{attribute 'pack_mode' := '2'}
TYPE U_XTS_TRANSPORT_CTRL :
UNION
  stCtrl              : ST_XTS_TRANSPORT_CTRL;
  byCtrl    AT %I*    : ARRAY[1..SIZEOF(ST_XTS_TRANSPORT_CTRL)] OF BYTE;
END_UNION
END_TYPE

(* stored: Version 1.1.0.1, ProductVersion 3.1.4026.12
   DUT U_XTS_TRANSPORT_CTRL: Id {deff15b8-09d4-48a2-8558-995eb04c3b99} *)
